INTERFACE I_Reset  EXTENDS I_StatusEx

METHOD Reset
VAR_INPUT
END_VAR
END_METHOD

END_INTERFACE

(* stored: Version 1.1.0.1
   Itf I_Reset: Id {b13e0a07-13fe-4130-92d2-b67a6bf512d3}
   Method Reset: Id {6de39cad-1884-4ec7-b494-38b114cd7658} *)
